// TIA Portal V16 export
// export: Created 2023-04-28T20:34:29.0022789Z, ExportSetting WithDefaults, DisplayName Totally Integrated Automation Portal, DisplayVersion V16, DisplayName TIA Portal Version Control Interface, DisplayVersion V16, DisplayName TIA Portal Openness, DisplayVersion V16, DisplayName STEP 7 Professional, DisplayVersion V16, DisplayName STEP 7 Safety, DisplayVersion V16, DisplayName WinCC Professional, DisplayVersion V16
FUNCTION "AnalogInputScaling" : Void   // FC1, LAD
{ S7_Optimized_Access := 'TRUE' }
VERSION : 0.1
// stored: AutoNumber true, IsIECCheckEnabled false, SetENOAutomatically false, UDAEnableTagReadback false
   VAR_INPUT
      RawInput : Int;
      MinValue : Int;
      MaxValue : Int;
   END_VAR
   VAR_OUTPUT
      AnalogOutput : Real;
   END_VAR
   VAR_TEMP
      TempNormValue : Real;
   END_VAR
   VAR CONSTANT
      MIN_VALUE : Int := 0;
      MAX_VALUE : Int := 27648;
   END_VAR
BEGIN

REGION Network 1
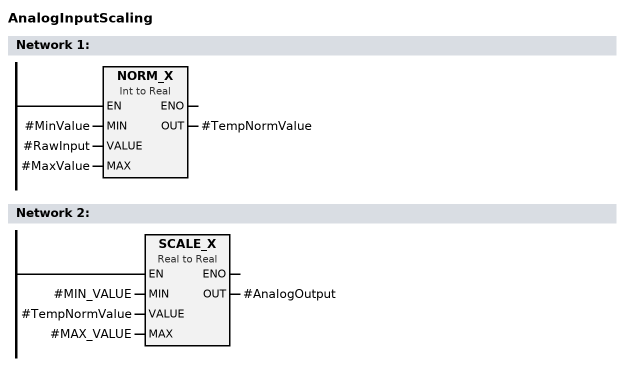
   RUNG wire#powerrail
      { S7_Templates := "[SrcType := Int, DestType := Real]" } Normalize(min := #MinValue, value := #RawInput, max := #MaxValue, out => #TempNormValue)
   END_RUNG
   // the same network as SCL:
   #TempNormValue := NORM_X(MIN := #MinValue, VALUE := #RawInput, MAX := #MaxValue);
END_REGION

REGION Network 2
   RUNG wire#powerrail
      { S7_Templates := "[SrcType := Real, DestType := Real]" } Scale(min := #MIN_VALUE, value := #TempNormValue, max := #MAX_VALUE, out => #AnalogOutput)
   END_RUNG
   // the same network as SCL:
   #AnalogOutput := SCALE_X(MIN := #MIN_VALUE, VALUE := #TempNormValue, MAX := #MAX_VALUE);
END_REGION
END_FUNCTION
